{attribute 'GeneratedUsingTerminal: EL3443-0000-0016'}
{attribute addProperty BoxType "EL3443-0000-0016"}
{attribute addProperty Id "Active_PowerAT %I*REAL4Apparent_PowerAT %I*REAL4Reactive_PowerAT %I*REAL4Power_FactorAT %I*REAL4"}
{attribute addProperty CRC "573578973"}
{attribute addProperty Size "16"}
TYPE L3_Power_22301EDD :
STRUCT
	{attribute addProperty Name "Active_Power"}
	Active_Power AT %I* : REAL;
	{attribute addProperty Name "Apparent_Power"}
	Apparent_Power AT %I* : REAL;
	{attribute addProperty Name "Reactive_Power"}
	Reactive_Power AT %I* : REAL;
	{attribute addProperty Name "Power_Factor"}
	Power_Factor AT %I* : REAL;
END_STRUCT
END_TYPE

(* stored: Version 1.2.0.0, ProductVersion 3.1.4024.9
   DUT L3_Power_22301EDD: Id {bfb02973-d2bf-48a1-a3e0-f47ca05c2d48} *)
